Staubli VAL3: RobotCfgStatus.dtx

public tool ExecuteTool = {fatherId=flange[0], ioLink=valve1}
public frame RefFrame = {fatherId=world[0]}
public num CyclePeriod
public mdesc MotionParm
